KUKA KRL program: chk_w9_rps2_opn.src

&ACCESS RVO4
&COMMENT Axor 903 Z2.1_Z2.2
DEF chk_w9_rps2_opn( )
; Check RPS AXOR 903 OPEN Z2.1/2
;//---- Start User-------

$TIMER[10] = 0
$TIMER_STOP[10] = FALSE

WAIT FOR (NOT $IN[498] AND NOT $IN[500])
WAIT FOR ($IN[497] AND $IN[499])

$TIMER_STOP[10] = TRUE
$TIMER[10] = 0

;//---- End User---------
END
